PROGRAM Collision_Detection
VAR
END_VAR

// NETWORK 1

ACTION High_Sensitivity:
// NETWORK 1
END_ACTION

END_PROGRAM

(* stored: Version 1.1.0.1, ProductVersion 3.1.4018.9
   POU Collision_Detection: Id {9ecdddc0-b25c-44ea-aec1-2464cfa2c870}, SpecialFunc None
   Action High_Sensitivity: Id {035d76ce-ea88-424a-9d56-ac3b4e9b0775} *)
